// TIA Portal V17 export
// export: Created 2025-05-06T14:49:43.3521464Z, ExportSetting WithDefaults, DisplayName Totally Integrated Automation Portal, DisplayVersion V17 Update 8, DisplayName TIA Portal Openness, DisplayVersion V17 Update 8, DisplayName TIA Portal Version Control Interface, DisplayVersion V17, DisplayName SINAMICS Startdrive Advanced, DisplayVersion V17 SP2, DisplayName SINAMICS Startdrive G110M, G120, G120C, G120D, G120P, G115D, DisplayVersion V17 SP2, DisplayName SINAMICS Startdrive G130, G150, S120, S150, SINAMICS MV, S210, DisplayVersion V17 SP2, DisplayName STEP 7 Professional, DisplayVersion V17 Update 8, DisplayName SINUMERIK ONE STEP 7 Toolbox, DisplayVersion V17 Update 12, DisplayName SINUMERIK 840D sl STEP 7 Toolbox, DisplayVersion V17 Update 12, DisplayName STEP 7 Safety, DisplayVersion V17 Update 6, DisplayName WinCC Advanced, DisplayVersion V17 Update 8
DATA_BLOCK "DB22109_HOPPER_1_UNIT_1_POWDER_FILLING_START_STOP_BY_CURRENT"   // DB22109
{ DB_Accessible_From_OPC_UA := 'FALSE' }
VERSION : 0.1
// stored: AutoNumber false, DBAccessibleFromOPCUA false, DBAccessibleFromWebserver true, InstanceOfName FB22108_POWDER_CURRENT_SENSOR, InstanceOfType FB
"FB22108_POWDER_CURRENT_SENSOR"
   // VAR_INPUT
   //    SENSOR_VALUE : Int;
   //    PF_LINE_ON : Bool;
   // END_VAR
   // VAR_OUTPUT
   //    CURRENT_LOW_LIMIT_ALARM : Bool;
   //    CURRENT_HIGH_LIMIT_ALARM : Bool;
   // END_VAR
   // VAR
   //    OUTPUT : Struct
   //       POWDER_FILLING_STOP_BY_CURRENT : Bool;
   //       POWDER_FILLING_START_BY_CURRENT : Bool;
   //    END_STRUCT;
   //    INPUT_SETTINGS : Struct
   //       NORMALIZED_VALUE : Real;
   //       SCALED_VALUE : Real;
   //    END_STRUCT;
   //    HMI : Struct
   //       HIGH_CURRENT_LIMIT : UInt;
   //       LOW_CURRENT_LIMIT : UInt;
   //    END_STRUCT;
   //    INTERNAL : Struct
   //       CURRENT_AVG_BLCK_START : Real;
   //       CURRENT_AVG_BLCK_STOP : Real;
   //       ACTUAL_CURRENT_TO_START : Real;
   //       ACTUAL_CURRENT_TO_STOP : Real;
   //    END_STRUCT;
   //    ALARM_SETTINGS : Struct
   //       ALARM_LOW_LIMIT : Real;
   //       ALARM_HIGH_LIMIT : Real;
   //    END_STRUCT;
   //    DB_CURRENT_AVERAGE_START : "FB22109_POWDER_CURRENT_AVG";
   //    DB_CURRENT_AVERAGE_STOP { S7_SetPoint := 'True'} : "FB22109_POWDER_CURRENT_AVG";
   //    START_BY_CURRENT_TIMER { S7_SetPoint := 'True'} : TON_TIME;
   //    CURRENT_HIGH_LIMIT_ALARM_TIMER { S7_SetPoint := 'True'} : TON_TIME;
   //    CURRENT_LOW_LIMIT_ALARM_TIMER { S7_SetPoint := 'True'} : TON_TIME;
   // END_VAR
BEGIN
END_DATA_BLOCK
